//Multiply
FUNCTION_BLOCK FB_2
VAR_INPUT
	nIn1:		INT;
	nIn2:		INT;
END_VAR
VAR_OUTPUT
	nOut1:		INT;
END_VAR
VAR
END_VAR

nOut1:=nIn1*nIn2;

END_FUNCTION_BLOCK

(* stored: Version 1.1.0.1, ProductVersion 3.1.4024.3
   POU FB_2: Id {9a850f11-b9b5-4216-a17a-e752cb2cd96f}, SpecialFunc None *)
